TYPE ST_VirtualHeatCounterDefaultParameters:
STRUCT
	tTaskCycleTime	: TIME;
	tCtrlCycleTime	: TIME;
END_STRUCT
END_TYPE

(* stored: Version 1.1.0.1, ProductVersion 3.1.4024.10
   DUT ST_VirtualHeatCounterDefaultParameters: Id {1d8d0424-1b08-450a-bbc7-3a6981abc718} *)
